FUNCTION_BLOCK EM_Check_Weigher IMPLEMENTS  ITF_EM_Check_Weigher
VAR_INPUT
END_VAR
VAR_OUTPUT
END_VAR
VAR
END_VAR

END_FUNCTION_BLOCK

(* stored: Version 1.1.0.1, ProductVersion 3.1.4024.12
   POU EM_Check_Weigher: Id {6a6823f3-6323-40e7-9859-29a8a1f5b7e8}, SpecialFunc None *)
